// TIA Portal project "Labview2" (V15)

(* hardware
DEVICE "S7-1200 station_1"  S7-1200 Station
   slot 0: "Rack_0"  S7-1200 Rack  Rack  V1.0
   slot 1: "PLC_1"  CPU 1214C DC/DC/DC  6ES7 214-1AG40-0XB0  V4.2
*)

// ===== PLC "PLC_1"  CPU 1214C DC/DC/DC =====

DATA_BLOCK "Bloque de datos_1"   // DB2
{ S7_Optimized_Access := 'TRUE' }
VERSION : 0.1
   VAR
      CONNECT : TCON_IP_v4;
      NDR : Bool;
      DR : Bool;
      ERROR : Bool;
      STATUS : Bool;
   END_VAR
BEGIN
   CONNECT.LocalPort := 502;
   CONNECT.InterfaceId := 64;
   CONNECT.ID := 1;
   CONNECT.ConnectionType := 11;
   CONNECT.RemoteAddress.ADDR[1] := 192;
   CONNECT.RemoteAddress.ADDR[2] := 168;
   CONNECT.RemoteAddress.ADDR[3] := 16#1;
   CONNECT.RemoteAddress.ADDR[4] := 100;
END_DATA_BLOCK

DATA_BLOCK "Bloque de datos_2"   // DB3
{ S7_Optimized_Access := 'TRUE' }
VERSION : 0.1
   VAR
      DATOS : Array[0..10] of Word;
   END_VAR
BEGIN
END_DATA_BLOCK

ORGANIZATION_BLOCK "Main"   // OB1, LAD, ProgramCycle
TITLE = "Main Program Sweep (Cycle)"
{ S7_Optimized_Access := 'TRUE' }
VERSION : 0.1
   VAR_INPUT
      Initial_Call : Bool;   // Initial call of this OB
      Remanence : Bool;   // =True, if remanent data are available
   END_VAR
BEGIN

REGION Network 1
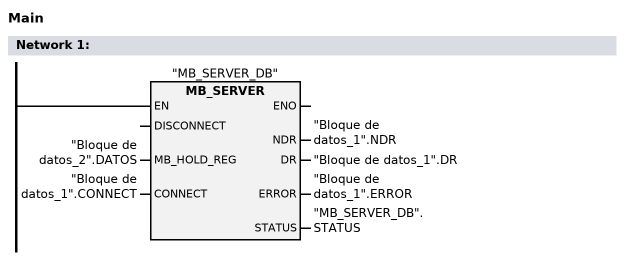
   "MB_SERVER_DB"(MB_HOLD_REG := "Bloque de datos_2".DATOS,   // MB_SERVER
                  CONNECT := "Bloque de datos_1".CONNECT,
                  NDR => "Bloque de datos_1".NDR,
                  DR => "Bloque de datos_1".DR,
                  ERROR => "Bloque de datos_1".ERROR,
                  STATUS => "MB_SERVER_DB".STATUS);
END_REGION
END_ORGANIZATION_BLOCK